// Mitsubishi GX Works2 project: De06   PLC: FX2N/FX2NC

PROGRAM MAIN
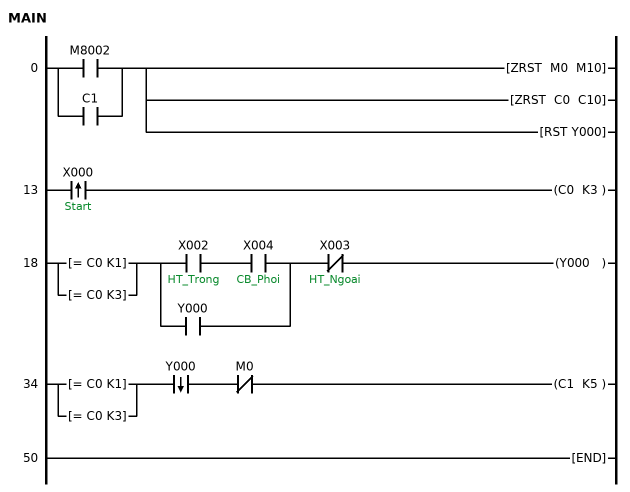
0     LD      M8002
      OR      C1
      ZRST    M0 M10
      ZRST    C0 C10
      RST     Y000
13    LDP     X000  ; Start
      OUT     C0 K3
18    LD=     C0 K1
      OR=     C0 K3
      LD      X002  ; HT_Trong
      AND     X004  ; CB_Phoi
      OR      Y000
      ANB
      ANI     X003  ; HT_Ngoai
      OUT     Y000
34    LD=     C0 K1
      OR=     C0 K3
      ANDF    Y000
      ANI     M0
      OUT     C1 K5
50    END
END_PROGRAM

// device comments not shown above
X001  ; Reset
